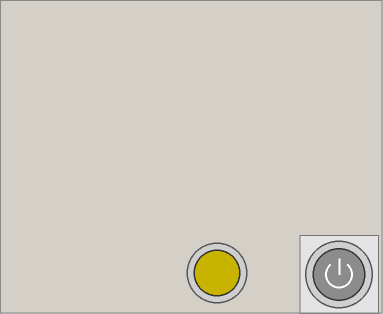
VISUALIZATION HMI_winch  // 383x314
    PowerSwitch (295,235 88x79), variable: GVL_HMIvars.stEnable.bWinchEnable, behaviour: TOGGLE, style: Switch-PowerSwitch-Gray
    Lamp1 (182,238 70x70), variable: GVL_HMIvars.stEnable.bWinchEnable, style: Lamp-Lamp1-Yellow
END_VISUALIZATION

(* stored: Version 1.1.0.1, ProductVersion 3.1.4024.12
   Visu HMI_winch: Id {1f09a1c1-b6c9-4f93-b207-fe691ee7c317} *)
